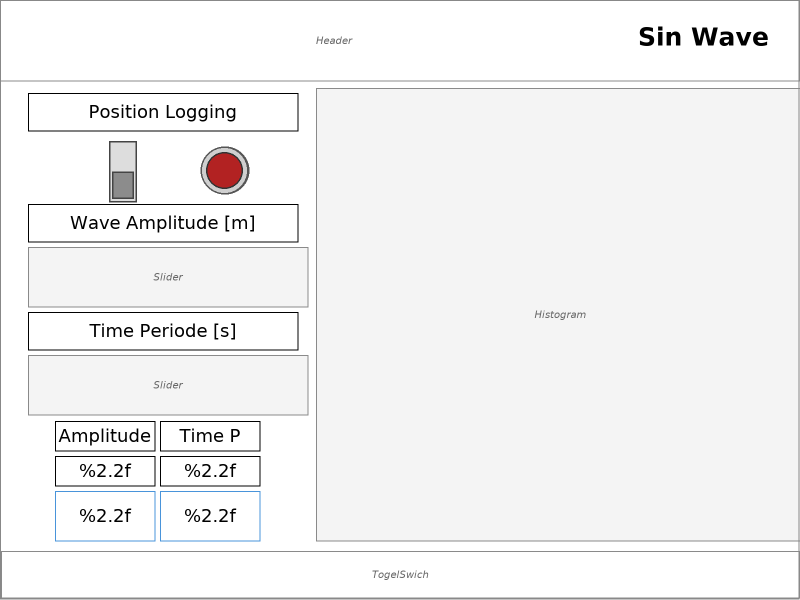
VISUALIZATION Visualization  // 800x600
    Frame (-132,0 932x81)
        shows Header()
    Frame (1,551 799x47)
        shows TogelSwich()
    Textfield (615,20 177x33), "Sin Wave"
    Histogram (316,88 489x453), scale format: %.1f, scale 1..2
        p1518820177: HMI.arrSinPayLoadPositions
        p102497268: HMI.arrSinPayLoadPositions
        p788070771: ARRAY [1..100] OF LREAL
    DipSwitch (54,141 138x61), variable: HMI.bSwichForPlot, behaviour: TOGGLE, style: Switch-DipSwitch-Gray
    Rectangle (28,93 270x38), "Position Logging", text variable: HMI.bData1
    Lamp1 (198,143 55x55), variable: HMI.bSwichForPlot, invisible if: not HMI.bSwichForPlot, style: Lamp-Lamp1-Green
    Lamp1 (197,143 55x55), variable: not HMI.bSwichForPlot, invisible if: HMI.bSwichForPlot, style: Lamp-Lamp1-Red
    Rectangle (55,491 100x50), "%2.2f", text variable: HMI.bAmplitudeWave
        OnMouseDown: write HMI.bAmplitudeWave via VisuDialogs.Numpad, min 0, max 40
    Rectangle (55,456 100x30), "%2.2f", text variable: HMI.bAmplitudeWave
    Rectangle (160,456 100x30), "%2.2f", text variable: HMI.bTimePriod
    Rectangle (160,491 100x50), "%2.2f", text variable: HMI.bTimePriod
        OnMouseDown: write HMI.bTimePriod via VisuDialogs.Numpad, min 0, max 40
    Rectangle (55,421 100x30), "Amplitude", text variable: HMI.bData1
    Rectangle (160,421 100x30), "Time P", text variable: HMI.bData1
    Rectangle (28,204 270x38), "Wave Amplitude [m]"
    Slider (28,247 280x60), variable: HMI.bAmplitudeWave, scale 0.1..2
    Rectangle (28,312 270x38), "Time Periode [s]"
    Slider (28,355 280x60), variable: HMI.bTimePriod, scale 5..105
END_VISUALIZATION

(* stored: Version 1.1.0.1, ProductVersion 3.1.4024.12
   Visu Visualization: Id {55b8d342-0396-40da-a9ce-c3a484582388} *)
